INTERFACE I_HostObjects

METHOD RegisterAbortable : HRESULT
VAR_INPUT
	Abortable : I_Abortable;
END_VAR
END_METHOD

METHOD RegisterCyclic : HRESULT
VAR_INPUT
	Cyclic : I_Cyclic;
END_VAR
END_METHOD

METHOD RegisterInitialisable : HRESULT
VAR_INPUT
	Initialisable : I_Initialisable;
END_VAR
END_METHOD

METHOD RegisterObject : HRESULT
VAR_INPUT
	Registerable : I_Object;
END_VAR
END_METHOD

METHOD RegisterResettable : HRESULT
VAR_INPUT
	Resetable : I_Resettable;
END_VAR
END_METHOD

METHOD RegisterTask : HRESULT
VAR_INPUT
	Task : I_Task;
END_VAR
END_METHOD

END_INTERFACE

(* stored: Version 1.1.0.1
   Itf I_HostObjects: Id {6b3f79ad-2a92-40cb-aed5-e9af4ed01870}
   Method RegisterAbortable: Id {be1b7b70-9d09-49cb-90c6-a693376757b0}
   Method RegisterCyclic: Id {80050db3-80e5-46b3-b147-b75b5f1ab81a}
   Method RegisterInitialisable: Id {7d5a17f2-c0ba-4781-8fb0-3013526db5cb}
   Method RegisterObject: Id {dd3d0223-46c8-4aa6-809a-31ad560b377a}
   Method RegisterResettable: Id {04daf7da-6efd-45f8-8b64-3bc15c24a64f}
   Method RegisterTask: Id {6638648b-69a5-453e-8b03-64c126ec6541} *)
